VAR_GLOBAL

END_VAR

(* stored: Version 1.1.0.1, ProductVersion 3.1.4024.9
   GVL GVL: Id {1baad497-2ec0-467b-a66f-b4b7960c6672} *)
